Staubli VAL3: Axis8Status.pgx

public program Axis8Status(bool& x_bPowerOn (dimensions=1), bool& x_bAlarm (dimensions=1), bool& x_bhome (dimensions=1))
begin
  //  x_bAlarm=true
  //  x_bPowerOn=false
  x_bhome=dDio["In4_b8BackHome"]==true
  x_bPowerOn=dDio["In4_b8MotorPower"]==true
  x_bAlarm=dDio["In4_b8MotorError"]==true


end
